FUNCTION_BLOCK FB_CommandAndControl
VAR_INPUT
END_VAR
VAR_OUTPUT
END_VAR
VAR
END_VAR

METHOD M_InitializeCounter
VAR_INPUT
END_VAR
END_METHOD

END_FUNCTION_BLOCK

(* stored: Version 1.1.0.1, ProductVersion 3.1.4024.9
   POU FB_CommandAndControl: Id {a2e6dd55-964d-4226-8a10-c1b60ea3b5a8}, SpecialFunc None
   Method M_InitializeCounter: Id {449694b4-695b-40c5-bd17-db12b965b5a7} *)
